FUNCTION_BLOCK FB_LightOffCommand IMPLEMENTS I_Command
VAR_INPUT
END_VAR
VAR_OUTPUT
END_VAR
VAR
	_rfbLight		: REFERENCE TO FB_Light;
END_VAR

METHOD execute : BOOL
_rfbLight.turnLightOff();
END_METHOD

//FB_Init is always available implicitly and it is used primarily for initialization.
//The return value is not evaluated. For a specific influence, you can also declare the
//methods explicitly and provide additional code there with the standard initialization
//code. You can evaluate the return value.
METHOD FB_Init: BOOL
VAR_INPUT
    bInitRetains: BOOL; // TRUE: the retain variables are initialized (reset warm / reset cold)
    bInCopyCode: BOOL;  // TRUE: the instance will be copied to the copy code afterward (online change)   
	rfbLight	:REFERENCE TO FB_Light;
END_VAR
_rfbLight REF= rfbLight;
END_METHOD

END_FUNCTION_BLOCK

(* stored: Version 1.1.0.1
   POU FB_LightOffCommand: Id {24e68c8e-25d3-4997-98ae-e7c2f4df045b}, SpecialFunc None
   Method execute: Id {19e333ec-461d-4314-b376-e7fa715a20cc}
   Method FB_Init: Id {0d49fddc-1181-4092-83ee-69feb0212b5f} *)
